FUNCTION_BLOCK EtherCatDevice EXTENDS SM_EtherCatDevice
VAR_INPUT
END_VAR
VAR_OUTPUT
END_VAR
VAR
    testVar : INT;
END_VAR

IF GLOBAL.CONFIG.SIMULATION_ACTIVE THEN
    SUPER^.infoData := 8;
    SUPER^.wcState := FALSE;
END_IF

SUPER^();

actualStatus := F_ConvStateToString(UINT_TO_WORD(infoData));

END_FUNCTION_BLOCK

(* stored: Version 1.1.0.1, ProductVersion 3.1.4018.2
   POU EtherCatDevice: Id {9c0828ff-c601-44f3-b01a-d1ae04f427f7}, SpecialFunc None *)
